(* PLC project Untitled1, Beckhoff Automation GmbH TF6420 Database Server Query Analyser 1.0.0.0 *)
(* stored: creationDateTime 2023-11-03T13:37:41, modificationDateTime 2023-11-03T13:37:41 *)

TYPE ST_Database_input : STRUCT
  power : REAL;
  test : REAL;
  time : REAL;
END_STRUCT;
END_TYPE
